(* CODESYS project set_in_mode.20190528.1.project

Project tree, tasks and I/O mapping:
  MIC7001 : Changsha Xiangji-ARM Cortex A9(xilinx zynq7000)-linux, Changsha Xiangji Hiden Technology Co.Ltd, version 3.5.10.40
    application Application
      libraries: Standard, * (System); CAA File, * (CAA Technical Workgroup); CAA Types Extern, * (CAA Technical Workgroup); CAA Callback Extern, * (CAA Technical Workgroup); SysMem, * (System); Util, 3.5.11.0 (System); SysFile, 3.5.9.0 (System); SysTypes Interfaces, * (System); CAN API, 1.0.0.3 (3S - Smart Software Solutions GmbH); SysTime, * (System); CAA DTUtil Extern, 3.5.12.0 (CAA Technical Workgroup); CAA SerialCom, 3.5.12.0 (CAA Technical Workgroup); cyber gpio, 3.5.10.40 (cyber); AC_DataLog, 3.5.13.0 (3S - Smart Software Solutions GmbH)
      task MainTask (cyclic, interval 20 ms, priority 15) calls prg_set_inmode
      program prg_set_inmode [ST]
      functions/
        function fn_write_in_mode_file [ST]
        function fn_read_in_mode_file [ST]
    SoftMotion General Axis Pool
    IoDrvMIC7001 : IoDrvMIC7001, Cyber-MI, version 19.1.1
        unmapped channels: Ai00@C16, Ai01@C28, Ai02@C17, Ai03@C29, Ai04@C30, Ai05@C19, Ai06@C31, Ai07@C20, Ai08@C18, Ai09@D18, Ai10@D20, Ai11@D31, Ai12@D19, Ai13@D30, Ai14@D29, Ai15@D17, Ai16@D28, Ai17@D16, Ai18-Do00@C25, Ai19-Do01@C24, Ai20-Do02@C13, Ai21-Do03@C01, Ai22-Do04@C03, Ai23-Do05@C04, Ai24-Do06@C05, Ai25-Do07@C06, Ai26-Do08@C08, Ai27-Do09@C09, Ai28-Do10@C10, Ai29-Do11@C11, Ai30-Do12@D34, Ai31-Do13@D35, Ai32-Do14@D23, Ai33-Do15@D12, Ai34-Do16@D10, Ai35-Do17@D09, Ai36-Do18@D08, Ai37-Do19@D07, Ai38-Do20@D05, Ai39-Do21@D04,
          Ai40-Do22@D03, Ai41-Do23@D02, Ai42-Do24@C23, Ai43-Do25@C35, Ai44-Do26@D24, Ai45-Do27@D13, Ai46-Ao00@C22, Ai47-Ao01@D14, Ai48_Pi02, Ai49_Out5V, Ai50_VCC, Ai51_VCC_L, Ai52_VCC_R, Ai53_Pwm-i0, Ai54_Pwm-i1, Ai55_Pwm-i2, Ai56_Pwm-i3, Ai57_CPU-T, Ai58_G-x, Ai59_G-y, Ai60_G-z, Ai61-reserved, Ai62-IO-cntr, Ai63-CDS-cntr, Di00-Ai00@C16, Di01-Ai01@C28, Di02-Ai02@C17, Di03-Ai03@C29, Di04-Ai04@C30, Di05-Ai05@C19, Di06-Ai06@C31, Di07-Ai07@C20, Di08-Ai08@C18, Di09-Ai09@D18, Di10-Ai10@D20, Di11-Ai11@D31, Di12-Ai12@D19, Di13-Ai13@D30, Di14-Ai14@D29, Di15-Ai15@D17,
          Di16-Ai16@D28, Di17-Ai17@D16, Di18-Ai18@C25, Di19-Ai19@C24, Di20-Ai20@C13, Di21-Ai21@C01, Di22-Ai22@C03, Di23-Ai23@C04, Di24-Ai24@C05, Di25-Ai25@C06, Di26-Ai26@C08, Di27-Ai27@C09, Di28-Ai28@C10, Di29-Ai29@C11, Di30-Ai30@D34, Di31-Ai31@D35, Di32-Ai32@D23, Di33-Ai33@D12, Di34-Ai34@D10, Di35-Ai35@D09, Di36-Ai36@D08, Di37-Ai37@D07, Di38-Ai38@D05, Di39-Ai39@D04, Di40-Ai40@D03, Di41-Ai41@D02, Di42-Ai42@C23, Di43-Ai43@C35, Di44-Ai44@D24, Di45-Ai45@D13, Di46-Ai46@C22, Di47-Ai47@D14, Di48-Pi00@C15, Di49-Pi01@C14, Di50-Pi02@D22, Di51-Pi03@D21, Di52-reserved, Di53-reserved, Di54-reserved, Di55-reserved,
          Di56-reserved, Di57-reserved, Di58-reserved, Di59-reserved, Di60-reserved, Di61-reserved, Di62-reserved, Di63-reserved, Pi00-Di48@C15, Pi01-Di49@C14, Pi02-Di50@D22, Pi03-Di51@D21, Do00-Ai18@C25, Do01-Ai19@C24, Do02-Ai20@C13, Do03-Ai21@C01, Do04-Ai22@C03, Do05-Ai23@C04, Do06-Ai24@C05, Do07-Ai25@C06, Do08-Ai26@C08, Do09-Ai27@C09, Do10-Ai28@C10, Do11-Ai29@C11, Do12-Ai30@D34, Do13-Ai31@D35, Do14-Ai32@D23, Do15-Ai33@D12, Do16-Ai34@D10, Do17-Ai35@D09, Do18-Ai36@D08, Do19-Ai37@D07, Do20-Ai38@D05, Do21-Ai39@D04, Do22-Ai40@D03, Do23-Ai41@D02, Do24-Ai42@C23, Do25-Ai43@C35, Do26-Ai44@D24, Do27-Ai45@D13,
          Do28-Pwmi00@C33, Do29-Pwmi01@C34, Do30-Pwmi02@D25, Do31-Pwmi03@D26, PWM00@C25, PWM01@C24, PWM02@C13, PWM03@C01, PWM04@C03, PWM05@C04, PWM06@C05, PWM07@C06, PWM08@C08, PWM09@C09, PWM10@C10, PWM11@C11, PWM12@D34, PWM13@D35, PWM14@D23, PWM15@D12, PWM16@D10, PWM17@D09, PWM18@D08, PWM19@D07, PWM20@D05, PWM21@D04, PWM22@D03, PWM23@D02, PWM24@C23, PWM25@C35, PWM26@D24, PWM27@D13, PWM28-Pwmi00@C33, PWM29-Pwmi01@C34, PWM30-Pwmi02@D25, PWM31-Pwmi03@D26, PWM_I_0@C33, PWM_I_1@C34, PWM_I_2@D25, PWM_I_3@D26,
          Ao00-Ai46@C22, Ao01-Ai47@D14, LED_run, LED_err, LED_usr, ctrl_ai_raw, ctrl_adjust, ctrl_adj0, ctrl_adj1, ctrl_adj2, ctrl_adj3, disable_5V
  text list GlobalTextList
*)

// MIC7001/Application/prg_set_inmode
PROGRAM prg_set_inmode
VAR
	stat:UINT := 0;
	old_in_mode:ARRAY[0..47] OF UINT;  //从已有文件中读出的配置
	in_mode:ARRAY[0..47] OF UINT;   //当前设定的配置
	number :UINT := 48;  //通道总数
	i: UINT;
	inmode_file:STRING:='in_mode.txt';
	
	MODE_0_5V :UINT := 0;
	MODE_0_36V :UINT := 1;
	MODE_0_20mA :UINT := 2;
	MODE_0_30Kohm :UINT := 3;
	MODE_DI_HIGH :UINT := 4;
	MODE_DI_LOW :UINT := 5;
END_VAR


CASE stat OF
0: //read inmode.txt
	IF fn_read_in_mode_file(pInMOde := ADR(old_in_mode), number := number) THEN
		stat := 50;
	ELSE 
		stat := 10;
	END_IF
10: //need write
	IF fn_write_in_mode_file(pInMode := ADR(in_mode), number := number) THEN
		stat := 100; //succeed
	END_IF

50: //the file inmode.txt is exist.
	FOR i := 0 TO number-1 DO
		IF old_in_mode[i] <> in_mode[i] THEN
			stat := 10; //write new config
			RETURN;
		END_IF
	END_FOR
	stat := 100;

100: //succeed, return;
	RETURN;
END_CASE

//默认全部设置为  0~5V输入
FOR  i := 0 TO number-1 DO
	in_mode[i] := 0;
END_FOR

//            上面的代码不用改动
//*********************************************************


//根据实际情况设置每个端口的类型
in_mode[0] := MODE_0_20mA;  //0~20 mA 
in_mode[1] := MODE_0_5V;  //默认为  MODE_0_5V， 可以不设置
in_mode[2] := MODE_0_36V;  
in_mode[3] := MODE_0_36V;
//.........
in_mode[47] := MODE_DI_LOW;   //最后一个

END_PROGRAM

// MIC7001/Application/functions/fn_read_in_mode_file
FUNCTION fn_read_in_mode_file : BOOL
VAR_INPUT
	pInMode :POINTER TO UINT;
	number:UINT;
END_VAR
VAR
	hFile: RTS_IEC_HANDLE;
	udiOpenError: RTS_IEC_RESULT;
	udiReadError: RTS_IEC_RESULT;
	i :DWORD;
	iTemp: UDINT;
	udiPos: UDINT;
	str: STRING(65535);
	str_size: __XWORD;
	udiByteRead: LWORD;

	len_of_line: INT;
	len_of_number :INT;
	magicNumber:REAL;
	check_sum:REAL:= 0;
	temp_num:REAL;
	index :UINT;
	mode: UINT;
END_VAR

fn_read_in_mode_file := FALSE;

//检测文件是否存在
hFile := sysfileopen(szFile := prg_set_inmode.inmode_file, am := sysfile.AM_READ, pResult:= ADR(udiOpenError));
IF hFile = RTS_INVALID_HANDLE	THEN  //文件不存在
	RETURN;
END_IF

//文件存在，开始读取内容
udiPos := SysFileSetPos(hFile:=hFile, ulOffset := 0);
udiByteRead := sysfile.SysFileRead(hfile := hFile,pbyBuffer := ADR(str), ulSize := SIZEOF(str), pResult := ADR(udiReadError));
IF udiByteRead < 1 THEN  //读取失败
	sysfile.SysFileClose(hFile := hFile);
	RETURN;
END_IF
sysfile.SysFileClose(hFile);

//读取本行的数字
FOR i := 0 TO number-1 DO
	len_of_number := find(str, '$N');
	mode := STRING_TO_UINT(left(str,len_of_number-1));
	str := delete(str, len_of_number,1);	
	pInMode[i] := mode;
END_FOR

fn_read_in_mode_file := TRUE;
RETURN;

END_FUNCTION

// MIC7001/Application/functions/fn_write_in_mode_file
FUNCTION fn_write_in_mode_file : BOOL
VAR_INPUT
	pInMode :POINTER TO UINT;
	number:UINT;
END_VAR
VAR
	bak_file_prefix:STRING :=ANY_TO_STRING("in_mode_bak_");
	bak_file:STRING := ANY_TO_STRING("");	
	hFile: RTS_IEC_HANDLE;
	udiDeleteError: RTS_IEC_RESULT;
	udiOpenError: RTS_IEC_RESULT;
	udiWriteError: RTS_IEC_RESULT;
	filesize: __XWORD;
	i :DWORD;
	iTemp: UDINT;
	udiPos: UDINT;
	str: STRING(256);
	str_size: __XWORD;
	udiByteWrite: LWORD;
	check_sum:REAL := 0;
END_VAR

fn_write_in_mode_file := FALSE;

IF number = 0 THEN
	RETURN;
END_IF

hFile := sysfileopen(szFile := prg_set_inmode.inmode_file, am := sysfile.AM_WRITE, pResult := ADR(udiOpenError));
IF hFile = RTS_INVALID_HANDLE THEN //创建文件失败
	RETURN;
END_IF
	
udiPos := SysFileSetPos(hFile:=hFile, ulOffset:=0);	
str:= ANY_TO_STRING('');
FOR i := 0 TO number-1 DO
	str := concat(str, ANY_TO_STRING(pInMode[i]));
	str := concat(str, '$N');	
END_FOR

str_size := ANY_TO_DWORD(len(str));
udiByteWrite := sysfile.SysFileWrite(hFile := hFile,pbyBuffer := ADR(str),ulSize := str_size, pResult := ADR(udiWriteError));

sysfile.SysFileClose(hFile);
fn_write_in_mode_file := TRUE;

END_FUNCTION
